Universal Robots PolyScope program: EGH80_grip.urp

Program EGH80_grip (installation=default directory=/programs createdIn=5.9.1.1031110 lastSavedIn=5.9.1.1031110 robotSerialNumber=20185500256)
Calibrated DH parameters: a=[0.000163, -0.146131, -0.38577, 0.000126, -0.000021, 0]; d=[0.161954, 188.306531, -157.478086, -30.695088, 0.099716, 0.099628]; alpha=[1.569701, -0.00212, 0.002263, 1.570438, -1.570123, 0]; deltaTheta=[0, -1.219859, 7.681919, -0.178877, -0.000001, 0]
Robot Program (runOnlyOnce=true)
  URCap EGH Grip (EGH-SCHUNK, SCHUNK GmbH & Co. KG) dataModel(actionType=true, pdTargetPosition=16.14, forceSave=6)
  Wait Sleep waitTime=1.5
  If EGH_is_success()≟ True  and EGH_is_endstop()≠ True
    URCap EGH Color Light band  (EGH-SCHUNK, SCHUNK GmbH & Co. KG)
    Script: return True
  Else 
    URCap EGH Color Light band  (EGH-SCHUNK, SCHUNK GmbH & Co. KG) dataModel(lb_color=Red)
    Script: return  False
